// TIA Portal V21 export
FUNCTION "Motore_PompaRicircoloAcquaCalda" : Void   // FC130, LAD
{ S7_Optimized_Access := 'TRUE' }
// stored: SetENOAutomatically false
   VAR_TEMP
      AutoPos : Bool;
      AutoNeg : Bool;
   END_VAR
BEGIN

REGION Network 1: Comando positivo in automatico
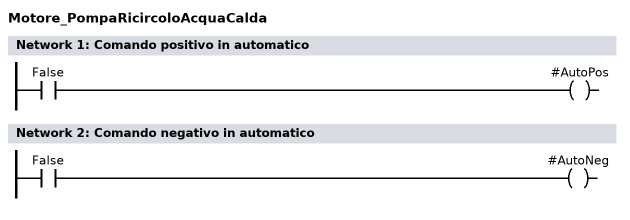
   RUNG wire#powerrail
      Contact( False )
      Coil( #AutoPos )
   END_RUNG
   // the same network as SCL:
   #AutoPos := False;
END_REGION

REGION Network 2: Comando negativo in automatico
   RUNG wire#powerrail
      Contact( False )
      Coil( #AutoNeg )
   END_RUNG
   // the same network as SCL:
   #AutoNeg := False;
END_REGION

REGION Network 3 (SCL)
   REGION PompaRicircoloAcquaCalda
       REGION Ingressi
           "Motore".M[K_Motore_PompaRicircoloAcquaCalda].In.FbDigitali.TermicoIntervenuto := NOT "PompaRicircoloAcqua_TermicoOk";
           "Motore".M[K_Motore_PompaRicircoloAcquaCalda].In.FbDigitali.FeedbackMarcia := "PompaRicircoloAcqua_Marcia";
           //"Motore".M["K_Motore_PompaRicircoloAcquaCalda"].In.CmdPosRich := #AutoPos;
           //"Motore".M["K_Motore_PompaRicircoloAcquaCalda"].In.CmdNegRich := #AutoNeg;
       END_REGION ;
       REGION Gestione
           "GestMotore"(K_Motore := "K_Motore_PompaRicircoloAcquaCalda",
                        K_TipoMotore := "K_TipoMotore_Teleruttore1Dir",
                        K_Zona := "K_Zona_Sterilizzatore");
       END_REGION ;
       REGION Uscite    
           "PompaRicircoloAcqua_ComandoMarcia" := "Motore".M[K_Motore_PompaRicircoloAcquaCalda].Out.CmdPosMotore;
       END_REGION ;
   END_REGION ;
END_REGION
END_FUNCTION
